(* CoDeSys 2.3 export: READINPUTS.EXP *)

(* POU InputsOutputs/ReadInputs, FBD *)
PROGRAM ReadInputs
VAR
	_input: ARRAY[0..11] OF INPUT;
END_VAR
VAR_OUTPUT
	IN0: BOOL;
	IN1: BOOL;
	IN2: BOOL;
	IN3: BOOL;
	IN4: BOOL;
	IN5: BOOL;
	IN6: BOOL;
	IN7: BOOL;
	IN8: BOOL;
	IN9: BOOL;
	IN10: BOOL;
	IN11: BOOL;
END_VAR
VAR CONSTANT
	ModeInput_Off: BYTE := 0;
	ModeInput_0_10V: BYTE := 3;
	ModeInput_Ratio: BYTE := 6;
	ModeInput_0_20mA: BYTE := 7;
	ModeInput_0_32V: BYTE := 9;
	ModeInput_LowSide: BYTE := 10;
	ModeInput_LowSideNamur: BYTE := 11;
	ModeInput_HighSide: BYTE := 12;
	ModeInput_Resistor: BYTE := 18;
END_VAR
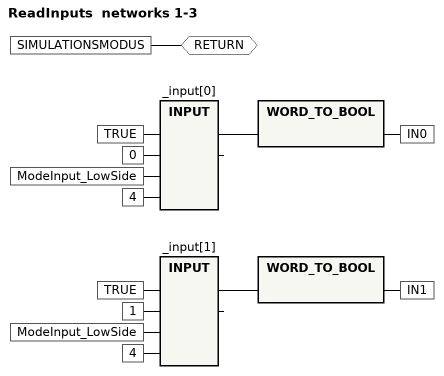
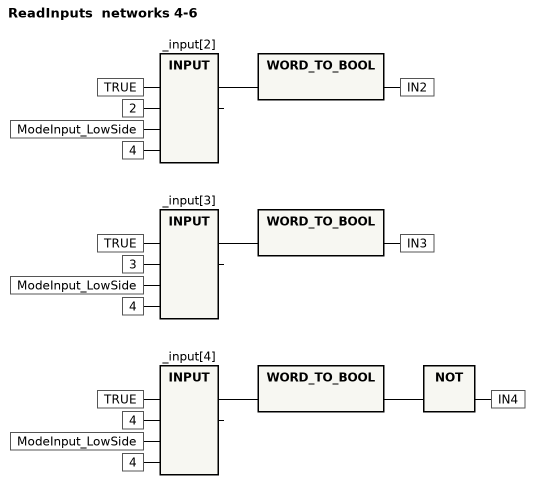
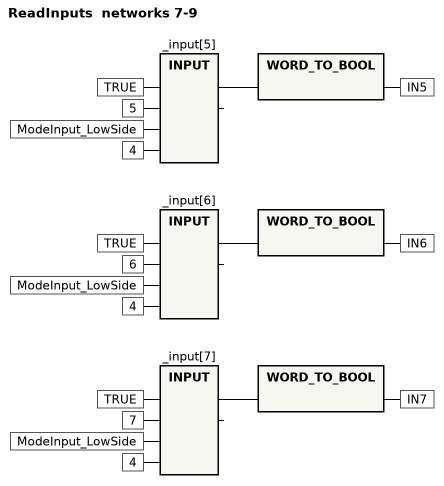
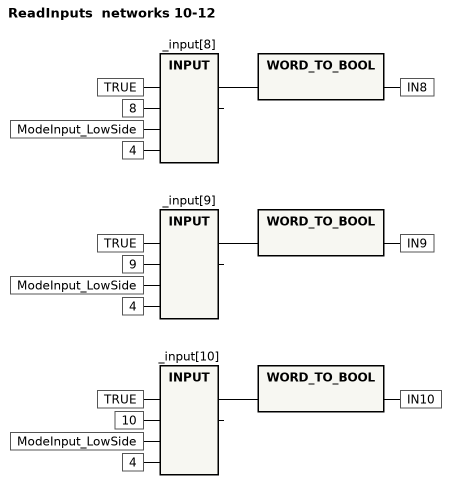
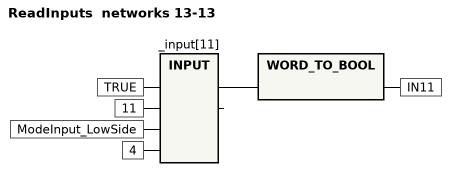
_FBD_ (* Function Block Diagram *)
NETWORK 1
	SIMULATIONSMODUS => <RETURN>
NETWORK 2
	WORD_TO_BOOL(_input[0]:INPUT(TRUE, 0, ModeInput_LowSide, 4)) => IN0
NETWORK 3
	WORD_TO_BOOL(_input[1]:INPUT(TRUE, 1, ModeInput_LowSide, 4)) => IN1
NETWORK 4
	WORD_TO_BOOL(_input[2]:INPUT(TRUE, 2, ModeInput_LowSide, 4)) => IN2
NETWORK 5
	WORD_TO_BOOL(_input[3]:INPUT(TRUE, 3, ModeInput_LowSide, 4)) => IN3
NETWORK 6
	NOT WORD_TO_BOOL(_input[4]:INPUT(TRUE, 4, ModeInput_LowSide, 4)) => IN4
NETWORK 7
	WORD_TO_BOOL(_input[5]:INPUT(TRUE, 5, ModeInput_LowSide, 4)) => IN5
NETWORK 8
	WORD_TO_BOOL(_input[6]:INPUT(TRUE, 6, ModeInput_LowSide, 4)) => IN6
NETWORK 9
	WORD_TO_BOOL(_input[7]:INPUT(TRUE, 7, ModeInput_LowSide, 4)) => IN7
NETWORK 10
	WORD_TO_BOOL(_input[8]:INPUT(TRUE, 8, ModeInput_LowSide, 4)) => IN8
NETWORK 11
	WORD_TO_BOOL(_input[9]:INPUT(TRUE, 9, ModeInput_LowSide, 4)) => IN9
NETWORK 12
	WORD_TO_BOOL(_input[10]:INPUT(TRUE, 10, ModeInput_LowSide, 4)) => IN10
NETWORK 13
	WORD_TO_BOOL(_input[11]:INPUT(TRUE, 11, ModeInput_LowSide, 4)) => IN11
_END_FBD_
END_PROGRAM
